// SIMATIC S7-200 project (STEP 7-Micro/WIN), CPU 224XP CN REL 02.01

ORGANIZATION_BLOCK MAIN:OB1
TITLE=PROGRAM COMMENTS
BEGIN
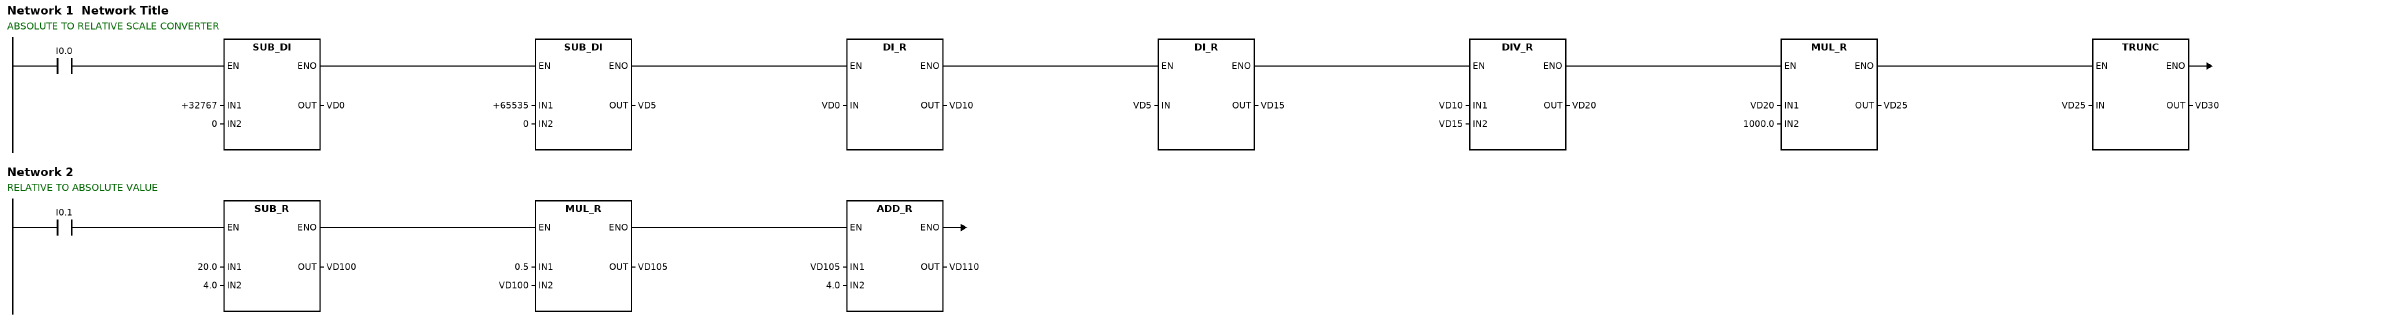
Network 1 // Network Title
// ABSOLUTE TO RELATIVE SCALE CONVERTER
LD     I0.0
MOVD   +32767, VD0
AENO
-D     0, VD0
AENO
MOVD   +65535, VD5
AENO
-D     0, VD5
AENO
DTR    VD0, VD10
AENO
DTR    VD5, VD15
AENO
MOVR   VD10, VD20
AENO
/R     VD15, VD20
AENO
MOVR   VD20, VD25
AENO
*R     1000.0, VD25
AENO
TRUNC  VD25, VD30
Network 2
// RELATIVE TO ABSOLUTE VALUE
LD     I0.1
MOVR   20.0, VD100
AENO
-R     4.0, VD100
AENO
MOVR   0.5, VD105
AENO
*R     VD100, VD105
AENO
MOVR   VD105, VD110
+R     4.0, VD110
END_ORGANIZATION_BLOCK
